{attribute 'qualified_only'}
{attribute 'strict'}
TYPE Antwort :
(
	pending,	//wartet auf Antwort
	timeout,
	ok,
	error,
	ignored,	//Ignore flag aktiviert
	expired		//Quittiert nach Error
);
END_TYPE

(* stored: Version 1.1.0.1, ProductVersion 3.1.4024.12
   DUT Antwort: Id {2de93a7a-8867-447f-bc81-c8ddcd1431da} *)
